// TIA Portal V17 export
// export: Created 2024-09-26T08:53:56.3591135Z, ExportSetting WithDefaults, DisplayName Totally Integrated Automation Portal, DisplayVersion V17, DisplayName TIA Portal Openness, DisplayVersion V17, DisplayName TIA Portal Version Control Interface, DisplayVersion V17, DisplayName STEP 7 Professional, DisplayVersion V17, DisplayName STEP 7 Safety, DisplayVersion V17, DisplayName WinCC Advanced / Unified PC, DisplayVersion V17
FUNCTION_BLOCK "SMA_Flow_1"   // FB2, LAD
{ S7_Optimized_Access := 'TRUE' }
VERSION : 0.1
// stored: AutoNumber true, IsIECCheckEnabled false, IsRetainMemResEnabled false, MemoryReserve 100, SetENOAutomatically false, UDAEnableTagReadback false
   VAR_INPUT
      bRun : Bool;
      tDutyCycle : Time;
      rFlow_Input : Real;
   END_VAR
   VAR_OUTPUT
      Flow { ExternalAccessible := 'False'; ExternalVisible := 'False'; ExternalWritable := 'False'} : Real;
   END_VAR
   VAR_TEMP
      bCount : Bool;
      bpulse1 : Bool;
      iCount : Int;
      aFlow : Array[0..200] of Real;
      i : Int;
   END_VAR
   VAR_TEMP   // added for the SCL form of the ladder/FBD networks
      _w1 : Bool;
      _w2 : Bool;
   END_VAR
BEGIN

REGION Network 1
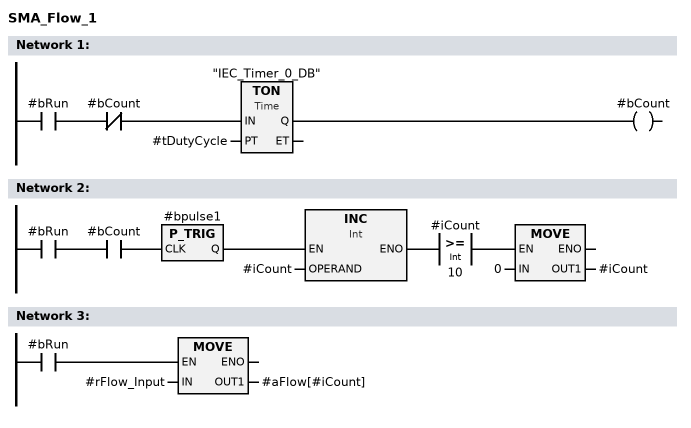
   RUNG wire#powerrail
      Contact( #bRun )
      I_Contact( #bCount )
      { S7_Templates := "time_type := Time" } "IEC_Timer_0_DB".TON(pt := #tDutyCycle, et =>)
      Coil( #bCount )
   END_RUNG
   // the same network as SCL:
   "IEC_Timer_0_DB".TON(IN := #bRun AND NOT #bCount, PT := #tDutyCycle);
   #bCount := "IEC_Timer_0_DB".Q;
END_REGION

REGION Network 2
   RUNG wire#powerrail
      Contact( #bRun )
      Contact( #bCount )
      P_Trig( #bpulse1 )
      { S7_Templates := "DestType := Int" } Inc( #iCount )
      { S7_Templates := "SrcType := Int" } GE_Contact(in1 := #iCount, in2 := 10)
      Move(in := 0, out1 => #iCount)
   END_RUNG
   // the same network as SCL:
   #_w1 := #bRun AND #bCount;
   #_w2 := #_w1 AND NOT #bpulse1;   // rising edge
   #bpulse1 := #_w1;
   IF #_w2 THEN #iCount := #iCount + 1; END_IF;
   IF #_w2 AND (#iCount >= 10) THEN #iCount := 0; END_IF;
END_REGION

REGION Network 3
   RUNG wire#powerrail
      Contact( #bRun )
      Move(in := #rFlow_Input, out1 => #aFlow[#iCount])
   END_RUNG
   // the same network as SCL:
   IF #bRun THEN #aFlow[#iCount] := #rFlow_Input; END_IF;
END_REGION

REGION Network 4 (SCL)
   FOR #i := 0 TO #iCount DO
       // Statement section FOR
       #Flow := #aFlow[#i] + #Flow;
       ;
   END_FOR;
END_REGION
END_FUNCTION_BLOCK
